INTERFACE ITF_HMI_PROVIDER

PROPERTY ItfHmiIn : REFERENCE TO ST_HMI_IN
GET
END_GET
END_PROPERTY

PROPERTY ItfHmiOut : REFERENCE TO ST_HMI_OUT
GET
END_GET
END_PROPERTY

/// reset
METHOD M_Reset : BOOL
VAR
END_VAR
END_METHOD

METHOD M_Run : BOOL
VAR_INPUT
END_VAR
END_METHOD

PROPERTY Mute : bool
GET
END_GET
END_PROPERTY

PROPERTY Provider : E_HMI_PROVIDER
GET
END_GET
END_PROPERTY

// HMI control request (Bedienhoheit)
//	set ti true, on any control request from the HMI provider (e.g.: watch IN struct)
//	reset will be done by HMI controller, on other provider request  
{attribute 'monitoring' := 'call'}
PROPERTY RequestManualControl : BOOL
GET
END_GET
SET
END_SET
END_PROPERTY

// HMI recipe control request (Bedienhoheit)  
{attribute 'monitoring' := 'call'}
PROPERTY RequestRecipeMgmt : BOOL
GET
END_GET
SET
END_SET
END_PROPERTY

// HMI settings control request (Bedienhoheit)  
{attribute 'monitoring' := 'call'}
PROPERTY RequestSettingMgmt : BOOL
GET
END_GET
SET
END_SET
END_PROPERTY

// HMI user management control request (Bedienhoheit)  
{attribute 'monitoring' := 'call'}
PROPERTY RequestUserMgmt : BOOL
GET
END_GET
SET
END_SET
END_PROPERTY

END_INTERFACE

(* stored: Version 1.1.0.1, ProductVersion 3.1.4024.12
   Itf ITF_HMI_PROVIDER: Id {219cc275-7f64-4fdb-8aff-67e9a5fc7b6f}
   Folder Methods: Id {3f82c239-638b-4502-ae9f-245315d37f17}
   Folder Properties: Id {1672e975-d0d2-45d3-8ab7-86355377e7b8}
   Property ItfHmiIn: Id {4575fe8e-efbe-482b-9fb4-b4c12d920b08}
   Get Get: Id {e06eb870-c282-4779-933b-b4837a6201f1}
   Property ItfHmiOut: Id {e7c6f1f0-70e7-4eef-8290-7b630e8838b3}
   Get Get: Id {fc47e092-cec2-44d7-b28b-e1da85417b72}
   Method M_Reset: Id {a79a26cf-e3c2-4b17-82fe-bb5169d8281b}
   Method M_Run: Id {3df8db0b-4176-4208-93c6-a86ea25db0d4}
   Property Mute: Id {e5b62302-90be-42b3-8957-8fae2a73c7ea}
   Get Get: Id {0e731040-0539-410e-ab66-257c065ea076}
   Property Provider: Id {86b7d6f5-f78e-4de8-8cee-a8d75d0db03b}
   Get Get: Id {3415edfc-7c99-4031-b744-1a902bd98ecd}
   Property RequestManualControl: Id {d9f3abc9-ff81-47c4-b965-a983658d5c2b}
   Get Get: Id {f20bc6a8-baaf-4052-a6d8-974bba438fff}
   Set Set: Id {6fae0697-6b4c-48ef-a3de-29bf357dae20}
   Property RequestRecipeMgmt: Id {92fdf764-9d13-47a7-bf09-372a42ba0bd7}
   Get Get: Id {9782190e-f1a4-4541-8562-7aadbf83759d}
   Set Set: Id {853f15e3-8019-4e3c-809a-3c3b9ad0c384}
   Property RequestSettingMgmt: Id {8871d424-3fa1-4e9b-9cb1-46ee1ff07e39}
   Get Get: Id {c4904e0f-eccd-4b11-a884-7c919ac9cb90}
   Set Set: Id {fd2e8bd7-6b35-411d-9b0d-95e534751b9f}
   Property RequestUserMgmt: Id {b606ec5d-7426-457d-8088-89da2a4e6156}
   Get Get: Id {09c4a8cb-7aea-4559-a164-164679e0354f}
   Set Set: Id {363db7a9-6c1e-4006-b5f9-2166500024b6} *)
